Staubli VAL3: whichObjectUsed.pgx

program whichObjectUsed(num x_nConvNum (dimensions=1), num& x_nInUse[] (dimensions=1), num& x_nError[] (dimensions=1))
begin
  // This program checks if there is an object in the queue of the
  // conveyor number passed as parameter
  //
  // Input Param
  //  x_nConvNum   : Conveyor number
  //
  // Output Param
  //  x_nInUse     : value of the next available object ID in the queue
  //        -1 --> No Part Available
  //      0..n --> ID of the object
  //
  //  x_nError      : Error code
  //      0    --> No error
  //      3    --> Invalid conveyor number
  //
  //----------------------------------------------------------------
  //
  x_nError=0
  switch x_nConvNum
    case 0
      call cnv0:whichObjectUsed(x_nInUse)
    break
    case 1
      call cnv1:whichObjectUsed(x_nInUse)
    break
    default
      x_nError=3
    break
  endSwitch
end
